FUNCTION_BLOCK FB_ControlBox
VAR_INPUT
	bRealControlBox : BOOL;
END_VAR
VAR_OUTPUT
END_VAR
VAR
	fbVirtualControlBox : FB_VirtualControlBox;
	fbRealControlBox : FB_RealControlBox;
	fbSelectedControlBox : I_ControlBox := fbVirtualControlBox;
	fbStatus : FB_Status;
END_VAR

IF NOT(bRealControlBox) THEN
	fbSelectedControlBox := fbVirtualControlBox;
	
	fbStatus(
		bOff := VirtualControlBox.stVirtualInputs.bOnSelector,
		bFault := FALSE,
		bStart := VirtualControlBox.stVirtualInputs.bStartButton,
		bStop := VirtualControlBox.stVirtualInputs.bStopButton,
		bRunning := Work.bRunning,
		eStatus => Work.eStatus
	);
	
	IF NOT(VirtualControlBox.stVirtualInputs.bOnSelector) THEN
			fbSelectedControlBox.ModeSelector(TRUE, FALSE, FALSE);  
	ELSIF VirtualControlBox.stVirtualInputs.bOnSelector AND NOT(VirtualControlBox.stVirtualInputs.bAutoSelector) THEN
			fbSelectedControlBox.ModeSelector(FALSE, TRUE, FALSE);  
	ELSIF VirtualControlBox.stVirtualInputs.bOnSelector AND VirtualControlBox.stVirtualInputs.bAutoSelector THEN	
			fbSelectedControlBox.ModeSelector(FALSE, FALSE, TRUE);  
	ELSE	
			fbSelectedControlBox.ModeSelector(FALSE, FALSE, FALSE);	
	END_IF
	
END_IF

// To do
IF bRealControlBox THEN
	fbSelectedControlBox := fbRealControlBox;
END_IF

END_FUNCTION_BLOCK

(* stored: Version 1.1.0.1, ProductVersion 3.1.4024.10
   POU FB_ControlBox: Id {23a5fbb3-746f-49da-9ce4-8057d9ad01ee}, SpecialFunc None *)
